(* Logix 5000 project; controller Start_Stop_Timer Emulate 5570 rev 30.12; software revision 30.01 *)

TASK MainTask (continuous, watchdog 500 ms) : MainProgram

MODULES
   Local : Emulate 5570 (ICP 2, rev 30.12)
END_MODULES

PROGRAM MainProgram   (* main routine MainRoutine *)
VAR
   Motor : BOOL;
   Power : BOOL;
   Start : BOOL;
   Stop : BOOL;
   Timer : TIMER := (PRE := 10000);
END_VAR

ROUTINE MainRoutine   (* ladder *)
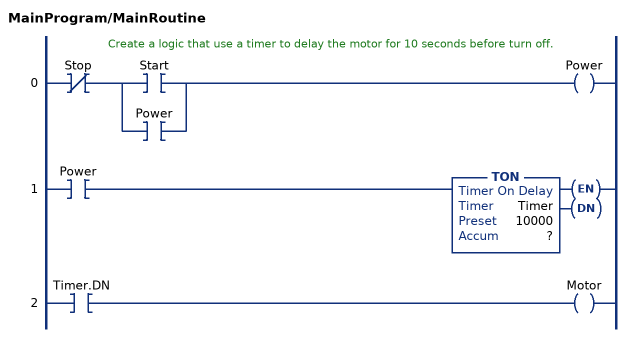
   // Create a logic that use a timer to delay the motor for 10 seconds before turn off.
   0: XIO(Stop)[XIC(Start) ,XIC(Power) ]OTE(Power);
   1: XIC(Power)TON(Timer,?,?);
   2: XIC(Timer.DN)OTE(Motor);
END_ROUTINE
END_PROGRAM
